FUNCTION_BLOCK T_TestRunner IMPLEMENTS I_TestRunner
VAR_INPUT
	TestSuiteName : T_MaxString := 'TestSuite';
    Verbose : BOOL;
END_VAR
VAR
    State : (
        sInit,
        sGetTest,
        sRunTest,
        sCheckResults
    );
    ResultsSummary   : T_MaxString;
    PassedTestsCount : DINT;
    FailedTestsCount : DINT;
    TestList         : T_ListOfTests(Capacity := 50);
    TestIterator     : T_TestIterator;
    CurrentTest      : I_UnitTest;

    RunTests      : BOOL := TRUE;
    TestFailed    : BOOL;
    TestCompleted : BOOL;
END_VAR

CASE State OF
    sInit:
        IF RunTests THEN
            RunTests := FALSE;
            TestIterator.Initialise(TestList);
            ResultsSummary   := '';
            FailedTestsCount := 0;
            PassedTestsCount := 0;
            F_LogResult(Source := TestSuiteName, Message := 'Starting Tests');
            State            := sGetTest;
        END_IF

    sGetTest:
        IF TestIterator.HasMore() THEN
            CurrentTest := TestIterator.GetNext();
            CurrentTest.Init();
            State := sRunTest;
        ELSE
            CurrentTest := 0;
            State       := sCheckResults;
        END_IF

    sRunTest:
        CurrentTest.RunTest(TestCompleted => TestCompleted,
                            TestFailed    => TestFailed);

        IF TestCompleted THEN
            IF TestFailed THEN
                FailedTestsCount := FailedTestsCount + 1;
                F_LogResult(Source := TestSuiteName, Message := FormatStringEx1('Test failed <%s>', CurrentTest.Name));
            ELSE
                PassedTestsCount := PassedTestsCount + 1;
                IF Verbose THEN
                    F_LogResult(Source := TestSuiteName, Message := FormatStringEx1('Test passed <%s>', CurrentTest.Name));
                END_IF
            END_IF
            State := sGetTest;
        END_IF

    sCheckResults:
        ResultsSummary := FormatString2('Tests completed. %d Tests Passed, %d Tests Failed',
                                          F_DINT(PassedTestsCount),
                                          F_DINT(FailedTestsCount));

        F_LogResult(Source  := TestSuiteName,
                    Message := FormatString2('Tests completed. %d Tests Passed, %d Tests Failed',
                                               F_DINT(PassedTestsCount),
                                               F_DINT(FailedTestsCount)));
        State := sInit;

END_CASE

METHOD AddTest
VAR_INPUT
    UnitTest : I_UnitTest;
END_VAR
TestList.AddTest(UnitTest);
END_METHOD

METHOD ClearTests
VAR_INPUT
END_VAR
TestList.Clear();
END_METHOD

{attribute 'call_after_online_change_slot' := '200'}
METHOD Start
VAR_INPUT
END_VAR
RunTests := TRUE;
END_METHOD

END_FUNCTION_BLOCK

(* stored: Version 1.1.0.1, ProductVersion 3.1.4024.12
   POU T_TestRunner: Id {c7f35beb-7079-466d-ae1a-1beb011dea9f}, SpecialFunc None
   Folder Methods: Id {35bbb33e-58f9-46f6-83b2-7eeb5a0d79dc}
   Method AddTest: Id {aff2d568-ab55-47bc-af2b-94e85ba5e218}
   Method ClearTests: Id {9c636768-dc92-4c10-a951-416ca0c5943a}
   Method Start: Id {78778059-eb1a-48b2-a0cc-e7bff17e395e} *)
